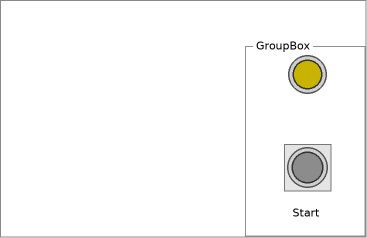
VISUALIZATION Visualization  // 367x238
    Lamp1 (285,52 45x45), variable: MAIN.bLamp, style: Lamp-Lamp1-Yellow
    PushSwitch (284,144 47x47), variable: MAIN.bStart, behaviour: TOGGLE, style: Switch-PushSwitch-Gray
    Label (277,198 58x30), "Start"
    GroupBox (245,38 120x198), "GroupBox"
END_VISUALIZATION

(* stored: Version 1.1.0.1, ProductVersion 3.1.4022.16
   Visu Visualization: Id {8cd9f448-2549-4088-8cbd-5cbee060cf77} *)
